PROGRAM MAIN
VAR
	
    bExecute1    : BOOL := FALSE;
	bExecute2    : BOOL := FALSE;
    nReadValue  : INT;           
    bBusy       : BOOL;
    bError      : BOOL;
    nErrId      : UDINT;
	sSymbol     : STRING := 'GVL_Config.nNumber';
	fbAdsRead1   : ADSRDWRTEX;
	fbAdsRead2   : ADSREAD;
	hVariable   : DWORD;
	
	fbRead1 : FB_Example1;
	fbRead2 : FB_Example2;
	fbWrite1 : FB_WriteExampl1;
	

END_VAR

IF bExecute1 THEN
	
	fbAdsRead1(
            NETID:= '', 
            PORT:= 852, 
            IDXGRP:= 16#F003,     
            IDXOFFS:= 0, 
            READLEN:= SIZEOF(hVariable),
			WRITELEN := INT_TO_UDINT(LEN(sSymbol)),
            SRCADDR:= ADR(sSymbol), 
            DESTADDR:= ADR(hVariable), 
            WRTRD:= TRUE, 
            BUSY => bBusy, ERR => bError, ERRID => nErrId);	
END_IF

IF bExecute2 THEN
	fbAdsRead2(
	NETID:= '', 
	PORT:= 852, 
	IDXGRP:= 16#F005 , 
	IDXOFFS:= hVariable, 
	LEN:= SIZEOF(nReadValue), 
	DESTADDR:= ADR(nReadValue), 
	READ:= bExecute2 , 
	BUSY => bBusy, 
	ERR => bError, 
	ERRID => nErrId);	
END_IF
fbRead1();
fbRead2();
fbWrite1();

END_PROGRAM

(* stored: Version 1.1.0.1, ProductVersion 3.1.4024.16
   POU MAIN: Id {db8aabc3-04c4-4f13-a554-30056803d64a}, SpecialFunc None *)
